// Mitsubishi GX Works2 project: WheelValveTapFX1S   PLC: FX1S

// global labels: Global1
VAR_GLOBAL
  XXPulse AT D8140 : DINT;
  YYPulse AT D8142 : DINT;
  YYTarget AT D4 : INT;
  YYFeed AT D6 : INT;
  XXTarget AT D0 : INT;
  XXFeed AT D2 : INT;
  YYRun AT M2 : BOOL;
  XXRun AT M0 : BOOL;
  XXMinI AT X002 : BOOL;
  XXMaxI AT X003 : BOOL;
  RunI AT X000 : BOOL;
  RunStopI AT X001 : BOOL;
  RunState AT D10 : INT;
  Run AT M10 : BOOL;
  RunStop AT M11 : BOOL;
  TapI AT X004 : BOOL;
  Tap AT M12 : BOOL;
  XXPulseO AT Y000 : BOOL;
  YYPulseO AT Y001 : BOOL;
  XXDirectionO AT Y004 : BOOL;
  YYDirectionO AT Y005 : BOOL;
  XXDirection AT M1 : BOOL;
  YYDirection AT M3 : BOOL;
END_VAR

// task Task_01 (event TRUE, interval 0, priority 31): POU_01

PROGRAM POU_01
VAR
  fStepReady : BOOL;
  fTmp : BOOL;
  fRise : BOOL;
  fRunStateNext : BOOL;
  fXXTarR : BOOL;
  fStepReadyTimerEN : BOOL;
END_VAR
SET(M8002, Y6);
MOV(M8002, 1000, XXFeed);
MOV(M8002, 1000, YYFeed);
(*|||||||||||||||*)
(*|||||||||||||||*)
SET(Run AND M100, fTmp);
MOV(fTmp, 2, RunState);
RST(fTmp, Run);
RST(fTmp, fTmp);
SET(RunStop, fTmp);
RST(fTmp, RunState);
RST(fTmp, XXRun);
RST(fTmp, YYRun);
RST(fTmp, fXXTarR);
RST(fTmp, fTmp);
(*|||||||||||||||*)
(*|||||||||||||||*)
DECO(TRUE, RunState, 4, M100);
(*|||||||||||||||*)
(*|||||||||||||||*)
OUT(NOT M8147 AND NOT M8148, fStepReadyTimerEN);
OUT_T(fStepReadyTimerEN, TC0, 1);
OUT(TC0, fStepReady);
(*move up*)
SET(fStepReady AND M102, fTmp);
RST(fTmp, XXDirection);
RST(fTmp, YYDirection);
SET(fTmp, XXRun);
SET(fTmp, YYRun);
SET(fTmp, fRunStateNext); RST(fTmp, fTmp);
(*move up done, ready*)
SET(fStepReady AND M103 AND fXXTarR, fTmp); RST(fTmp, fXXTarR);
SET(fTmp, fRunStateNext); RST(fTmp, fTmp);
(*wait tap hit, move down*)
SET(fStepReady AND M104 AND Tap, fTmp); RST(Tap, Tap);
SET(fTmp, XXDirection);
SET(fTmp, YYDirection);
SET(fTmp, XXRun);
SET(fTmp, YYRun);
SET(fTmp, fRunStateNext); RST(fTmp, fTmp);
(*move down done, move up*)
SET(fStepReady AND M105 AND fXXTarR, fTmp); RST(fTmp, fXXTarR);
RST(fTmp, XXDirection);
RST(fTmp, YYDirection);
SET(fTmp, XXRun);
SET(fTmp, YYRun);
SET(fTmp, fRunStateNext); RST(fTmp, fTmp);
(*move down done, return wait tap hit*)
SET(fStepReady AND M106 AND fXXTarR, fTmp); RST(fTmp, fXXTarR);
MOV(fTmp, 4, RunState); RST(fTmp, fTmp);
(*|||||||||||||||*)
(*|||||||||||||||*)
PLSY(XXRun, XXFeed, 0, XXPulseO);
RST(M8029, XXRun);
OUT(XXDirection, XXDirectionO);
RST(XXDirection AND XXMaxI, XXRun);
RST(NOT XXDirection AND XXMinI, XXRun);
PLF(XXRun, fRise); SET(fRise, fXXTarR);
(*|||||||||||||||*)
PLSY(YYRun, YYFeed, 0, YYPulseO);
RST(M8029, YYRun);
OUT(YYDirection, YYDirectionO);
RST(XXRun, YYRun);
(*|||||||||||||||*)
(*|||||||||||||||*)
PLS(RunI, fRise); SET(fRise, Run);
PLS(RunStopI, fRise); SET(fRise, RunStop);
PLS(TapI, fRise); SET(fRise, Tap);
(*|||||||||||||||*)
(*|||||||||||||||*)
INC(fRunStateNext, RunState); RST(fRunStateNext, fRunStateNext);
END_PROGRAM
